// TwinCAT 3 PLC project cooling
// ProgramVersion: 3.1.4022.7
// libraries:
//   Tc2_MC2, * (Beckhoff Automation GmbH)
//   Tc2_Standard, * (Beckhoff Automation GmbH)
//   Tc2_System, * (Beckhoff Automation GmbH)
//   Tc3_Module, * (Beckhoff Automation GmbH)
// project tree:
//   / PlcTask.TcTTO
//   POUs/ MAIN.TcPOU
// real-time tasks:
//   TASK PlcTask: cycle T#10ms, priority 20, ADS port 350
// motion (NC):
// I/O:
//   DEVICE Device 1 (EtherCAT), AmsNetId 172.21.148.24.2.1
//     Term 9 (EK1200)
// variable links:
//   cooling Instance <-> Device 1 (EtherCAT)/Term 10 (EK1200)/Term 3 (EL7047)
//     PlcTask Inputs/MAIN.extended <-> STM Status/Status/Digital input 2
//     PlcTask Inputs/MAIN.retracted <-> STM Status/Status/Digital input 1
//   cooling Instance <-> Device 1 (EtherCAT)/Term 10 (EK1200)/Term 8 (EL3064)
//     PlcTask Inputs/MAIN.i_iDistance_R <-> AI Standard Channel 1/Value
//     PlcTask Inputs/MAIN.i_irefV_R <-> AI Standard Channel 2/Value
//   cooling Instance <-> NC-Task 1 SAF/Axes/Axis 2
//     PlcTask Inputs/MAIN.axis.NcToPlc <-> Outputs/ToPlc
//     PlcTask Outputs/MAIN.axis.PlcToNc <-> Inputs/FromPlc

CONFIGURATION cooling
    RESOURCE PLC ON TwinCAT3
        TASK PlcTask(INTERVAL := T#10ms, PRIORITY := 20);
        PROGRAM MAIN WITH PlcTask : MAIN;
    END_RESOURCE
END_CONFIGURATION

// ---- POUs/MAIN.TcPOU
PROGRAM MAIN
VAR
	axis: AXIS_REF;
	iTermBits: DINT;
	rV : Real;
	i_iDistance_R AT %I* :DINT;
	rVref : Real;
	i_irefV_R AT %I* :DINT;
	power: MC_POWER;
	retracted AT %I* : BOOL;
	extended At %I* :BOOL;
END_VAR

//axis.ReadStatus();
iTermBits := DINT#16#7FFFFFFF;
rV := 10*DINT_TO_REAL(i_iDistance_R)/iTermBits;
rVref := 10*DINT_TO_REAL(i_irefV_R)/iTermBits;

power(Axis:=axis, Enable_Positive := NOT retracted, Enable_Negative:= NOT extended);

END_PROGRAM
